// TIA Portal project "OPC_UA_Example" (V14)

(* hardware
DEVICE "S71500/ET200MP-Station_1"  S7-1500 station
   slot 0: "Profilschiene_0"  Rack  6ES7 590-1***0-0AA0
   slot 1: "PLC_1"  CPU 1511C-1 PN  6ES7 511-1CK00-0AB0  V2.1
      slot 3: "CPU-Display_1"  6ES7591-1AA00-0AA0
*)

// ===== PLC "PLC_1"  CPU 1511C-1 PN =====

DATA_BLOCK "OPC_Variable_DB"   // DB1
{ S7_Optimized_Access := 'TRUE' }
VERSION : 0.1
// stored: InstanceOfName OPC_Variable
"OPC_Variable"
BEGIN
END_DATA_BLOCK

FUNCTION_BLOCK "OPC_Variable"   // FB1, SCL
{ S7_Optimized_Access := 'TRUE' }
VERSION : 0.1
   VAR
      OPC_Datein : Struct
         bV : Bool;
         IV : Int;
         SV : String;
      END_STRUCT;
   END_VAR
BEGIN
END_FUNCTION_BLOCK

ORGANIZATION_BLOCK "Main"   // OB1, LAD, ProgramCycle
TITLE = "Main Program Sweep (Cycle)"
{ S7_Optimized_Access := 'TRUE' }
VERSION : 0.1
   VAR_INPUT
      Initial_Call : Bool;   // Initial call of this OB
      Remanence : Bool;   // =True, if remanent data are available
   END_VAR
BEGIN

REGION Network 1
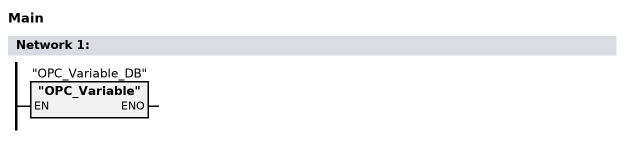
   RUNG wire#powerrail
      "OPC_Variable_DB"()
   END_RUNG
   // the same network as SCL:
   "OPC_Variable_DB"();   // "OPC_Variable"
END_REGION
END_ORGANIZATION_BLOCK